(* CoDeSys 2.3 export: MODBUSCONTROL.EXP *)

(* POU Modbus/ModbusControl, ST *)
PROGRAM ModbusControl
VAR_TEMP
	i: USINT;
END_VAR
(*чтение регистров Modbus*)
getModbusRegisters();

(*запись регистров Modbus*)
setModbusRegisters();
END_PROGRAM
